TYPE ST_ADJNODE :
STRUCT
	nNode	: INT;
	nWeight	: POINTER TO INT;
END_STRUCT
END_TYPE

(* stored: Version 1.1.0.1, ProductVersion 3.1.4024.12
   DUT ST_ADJNODE: Id {f8ab38e0-f2dc-4d52-ac01-6ec2e12194f3} *)
